// Provies interface to properties required for file access
INTERFACE I_FileProperties

// Gets or set file properties.
PROPERTY FileProperties : REFERENCE TO ST_FileProperties
GET
END_GET
SET
END_SET
END_PROPERTY

END_INTERFACE

(* stored: Version 1.1.0.1, ProductVersion 3.1.4024.13
   Itf I_FileProperties: Id {48c6fead-5114-0488-0fb4-ef75ebc9ec47}
   Property FileProperties: Id {ec9861a9-4e32-0443-1bd2-a47790c96b07}
   Get Get: Id {fde9c63d-afb5-0ac9-15c2-ddc3e531f4a7}
   Set Set: Id {58f44111-772d-080a-1c3c-93f51a0fd80d} *)
